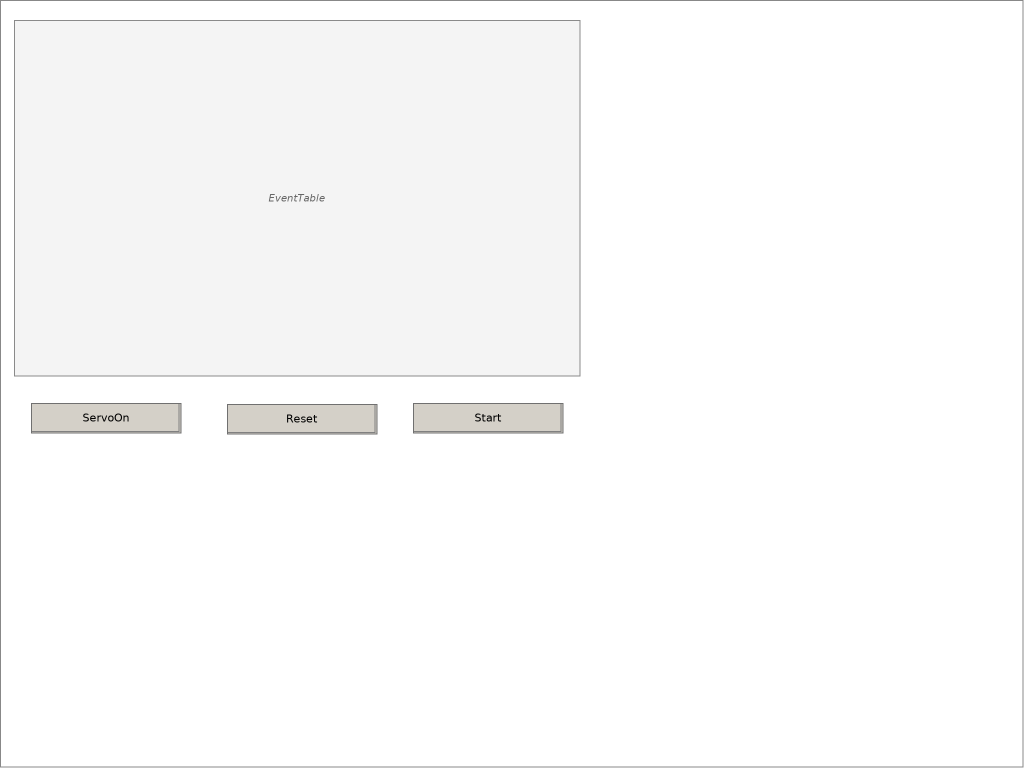
VISUALIZATION Visualization  // 1024x768
    EventTable (14,20 566x356)
        p1690906150: Class
        p3258520714: Date
        p2231227367: Time
        p3993844394: Message
        p2076579579: Details
        p3558512729: MAIN.Events.aEvents
        p3921149237: m_pDataArray..pArray
    Button (31,403 150x30), "ServoOn", pressed state: MAIN.ServoPower.Status
        toggle MAIN.ServoPower.Enable
    Button (413,403 150x30), "Start", pressed state: MAIN.control.McOutputs.Busy
        tap MAIN.control.Start
    Button (227,404 150x30), "Reset", pressed state: MAIN.ServoReset.Done
        tap MAIN.ServoReset.Execute
END_VISUALIZATION

(* stored: Version 1.1.0.1, ProductVersion 3.1.4024.9
   Visu Visualization: Id {28316d9f-6f8d-4738-bc51-42449769f597} *)
